FUNCTION_BLOCK RejectWithMessageSyncHandler IMPLEMENTS I_SynchronousRpcHandler
VAR
END_VAR

METHOD Handle
VAR_INPUT
	Parameters : I_Deserializer;
	Response : I_SynchronousRpcResponse;
END_VAR
VAR
END_VAR
Response.RejectWithError('EXAMPLE_ERROR_CODE','This is the reject message');
END_METHOD

END_FUNCTION_BLOCK

(* stored: Version 1.1.0.1, ProductVersion 3.1.4024.15
   POU RejectWithMessageSyncHandler: Id {4abf70fc-ce4e-4c80-b47e-9d4c86f97df6}, SpecialFunc None
   Method Handle: Id {716ba058-8390-49db-b2a1-86a7673c1055} *)
